PROGRAM BH0LPL_LineBackground
VAR
END_VAR

MAIN.stLine_BH0LPL.fbLine(stLine:=MAIN.stLine_BH0LPL);
MAIN.stLine_BH0LPL.stStation_BH0LPL01.fbStation(
				stLine:=MAIN.stLine_BH0LPL,
				stStation:=MAIN.stLine_BH0LPL.stStation_BH0LPL01);

END_PROGRAM

(* stored: Version 1.1.0.1, ProductVersion 3.1.4024.15
   POU BH0LPL_LineBackground: Id {dc4e4609-871f-448f-bdf3-6ff8783d59ff}, SpecialFunc None *)
